FUNCTION Convert_LWORD_TO_ULINT : Hresult
VAR_INPUT
	in : LWORD;
	out : REFERENCE TO ULINT;
END_VAR
VAR
	converted : ULINT;
END_VAR
VAR CONSTANT
	INCOMPATIBLE : HRESULT := 16#9811070E;
END_VAR

converted := LWORD_TO_ULINT(in);

IF (ULINT_TO_LWORD(converted) <> in) THEN
	Convert_LWORD_TO_ULINT := INCOMPATIBLE;
	RETURN;
END_IF

out := converted;

END_FUNCTION

(* stored: Version 1.1.0.1, ProductVersion 3.1.4024.12
   POU Convert_LWORD_TO_ULINT: Id {cf51b67d-c1f7-40c3-bc8e-581b06276ee4}, SpecialFunc None *)
